SUBAPPLICATION DecoratorDemo (* Decorator pattern demo: E_PERMIT gates TrueUntil.TRIGGER without modifying TrueUntil itself *)
  (* Standard: 61499-2; Description: Copyright (c) 2026 Meisterschulen am Ostbahnhof This program and the accompanying materials are made available under the terms of the Eclipse Public License 2.0 which is available at https://www.eclipse.org/legal/epl-2.0/ SPDX-License-Identifier: EPL-2.0 *)
  (* Version 1.0, 2026-08-31, Franz Höpfinger, Meisterschulen am Ostbahnhof, Decorator design pattern (IEC 61499 primer course, Module 6, Valeriy Vyatkin, slide 68), demo application *)
  PACKAGE Meins::DesingPatterns::DecoratorPattern;
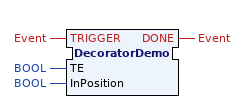
  EVENT_INPUT
    TRIGGER; (* Ask the step to run - only actually runs while TE is TRUE *)
  END_EVENT
  EVENT_OUTPUT
    DONE; (* The step completed (only fires if TE was TRUE when TRIGGER arrived) *)
  END_EVENT
  VAR_INPUT
    TE : BOOL := TRUE; (* Decorator condition: TRIGGER only reaches the step while this is TRUE *)
    InPosition : BOOL; (* Demo: simulate the step's actuator reaching its position *)
  END_VAR
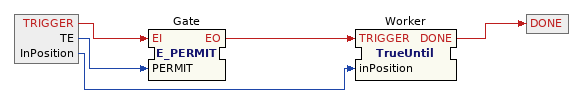
  FBS
    Gate : iec61499::events::E_PERMIT;
    Worker : Meins::DesingPatterns::ChainOfActionsPattern::TrueUntil;
  END_FBS
  EVENT_CONNECTIONS
    TRIGGER TO Gate.EI;
    Gate.EO TO Worker.TRIGGER;
    Worker.DONE TO DONE;
  END_CONNECTIONS
  DATA_CONNECTIONS
    TE TO Gate.PERMIT;
    InPosition TO Worker.inPosition;
  END_CONNECTIONS
END_SUBAPPLICATION
